// TIA Portal V18 export
DATA_BLOCK "Heatercontrol"   // DB140
{ S7_Optimized_Access := 'TRUE' }
VERSION : 0.1
// stored: AutoNumber true, DBAccessibleFromOPCUA true, IsOnlyStoredInLoadMemory false, IsRetainMemResEnabled false, IsWriteProtectedInAS false, MemoryReserve 100
   VAR RETAIN
      ON : Struct
         heater1 : Bool;
         heater2 : Bool;
         heater3 : Bool;
         heater4 : Bool;
      END_STRUCT;
      "heater ON HMI" : Bool;
   END_VAR
   VAR
      "Show heater Button" : Bool;
   END_VAR
BEGIN
END_DATA_BLOCK
